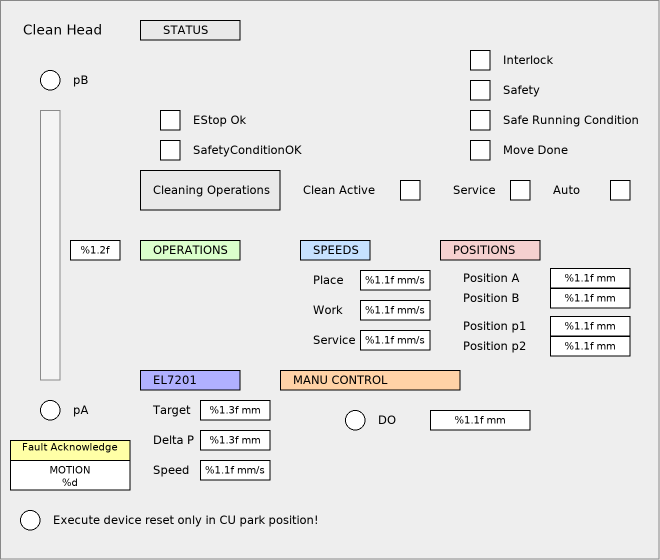
VISUALIZATION _VISU_CLEAN_CH  // 660x560
VAR_IN_OUT
  m_Inst : INT;               (*visu instance*) 
END_VAR
    Rectangle (0,0 660x560)
    Polyline (210,380)
    Polyline (510,250)
    Polyline (300,250)
    Rectangle (280,370 180x20)
    Rectangle (300,240 70x20)
    Rectangle (440,240 100x20)
    Rectangle (140,240 100x20)
    Rectangle (70,400 40x20), "pA"
    Ellipse (40,400 20x20), colour toggle: PRG_MACHINE.fb_CleaningCH[m_Inst].bL_Sensor_pA
    Ellipse (40,70 20x20), colour toggle: PRG_MACHINE.fb_CleaningCH[m_Inst].bI_Sensor_pB
    Rectangle (70,70 50x20), "pB"
    Rectangle (70,240 50x20), "%1.2f", text variable: 1000 * PRG_MACHINE.fb_CleaningCH[m_Inst].fB_Axis.fO_ActualPosition
    Rectangle (375,410 40x20), "DO"
    Rectangle (290,370 170x20), "MANU CONTROL"
    Polyline (450,380)
    Rectangle (310,240 70x20), "SPEEDS"
    Rectangle (360,270 70x20), "%1.1f mm/s", text variable: PRG_MACHINE.fb_CleaningCH[m_Inst].sI_SpeedDef.fP_PlaceSpeed
        OnMouseDown: write the text variable via VisuDialogs.Numpad
    Rectangle (360,300 70x20), "%1.1f mm/s", text variable: PRG_MACHINE.fb_CleaningCH[m_Inst].sI_SpeedDef.fP_WorkSpeed
        OnMouseDown: write the text variable via VisuDialogs.Numpad
    Rectangle (360,330 70x20), "%1.1f mm/s", text variable: PRG_MACHINE.fb_CleaningCH[m_Inst].sI_SpeedDef.fP_ServiceSpeed
        OnMouseDown: write the text variable via VisuDialogs.Numpad
    Rectangle (310,270 60x20), "Place"
    Rectangle (310,300 60x20), "Work"
    Rectangle (310,330 60x20), "Service"
        OnMouseDown: write the text variable via Edit
    Rectangle (550,268 80x20), "%1.1f mm", text variable: PRG_MACHINE.fb_CleaningCH[m_Inst].fI_Position_A
        OnMouseDown: write the text variable via VisuDialogs.Numpad
    Rectangle (460,268 85x20), "Position A"
    Rectangle (460,288 85x20), "Position B"
    Rectangle (550,288 80x20), "%1.1f mm", text variable: PRG_MACHINE.fb_CleaningCH[m_Inst].fI_Position_B
        OnMouseDown: write the text variable via VisuDialogs.Numpad
    Rectangle (450,240 90x20), "POSITIONS"
    Polyline (210,250)
    Rectangle (150,240 90x20), "OPERATIONS"
    Scrollbar (40,110 20x270)
        p3598130195: PRG_MACHINE.sADS_CleanAxis[iCPr_MAP_Cp_ChAxis[m_Inst]].sO_AxisPosition.fC_Min
        p2245068023: PRG_MACHINE.sADS_CleanAxis[iCPr_MAP_Cp_ChAxis[m_Inst]].sO_AxisPosition.fC_Max
        p1057716461: PRG_MACHINE.fb_CleaningCH[m_Inst].fB_Axis.fO_ActualPosition * 1000
    Ellipse (345,410 20x20), colour toggle: PRG_MACHINE.sADS_CleanAxis[iCPr_MAP_Cp_ChAxis[m_Inst]].bI_ManualMove, input disabled if: NOT PRG_MACHINE.sADS_CleanAxis[iCPr_MAP_Cp_ChAxis[m_Inst]].bO_ManualMoveCanEx
        toggle PRG_MACHINE.sADS_CleanAxis[iCPr_MAP_Cp_ChAxis[m_Inst]].bI_ManualMove
    Rectangle (20,20 120x20), "Clean Head"
    Rectangle (140,370 100x20)
    Rectangle (150,460 70x20), "Speed"
    Rectangle (200,460 70x20), "%1.1f mm/s", text variable: 1000 * PRG_MACHINE.fb_CleaningCH[m_Inst].fB_Axis.fI_SpeedLimit
    Rectangle (150,370 90x20), "EL7201"
    Rectangle (10,440 120x50), "Fault Acknowledge", colour toggle: (PRG_MACHINE.fb_CleaningCH[m_Inst].wL_ErrorCode) <> 0
    Polyline (130,450)
    RoundedRectangle (10,460 120x30), "%d", text variable: PRG_MACHINE.fb_CleaningCH[m_Inst].wL_ErrorCode
        tap PRG_MACHINE.sADS_CleanAxis[iCPr_MAP_Cp_ChAxis[m_Inst]].bI_FaultAck
    RoundedRectangle (40,460 60x20), "MOTION"
    Rectangle (140,170 140x40)
    Rectangle (140,20 100x20)
    Polyline (140,30)
    Polyline (240,30)
    Rectangle (160,20 60x20), "STATUS"
    RoundedRectangle (160,110 20x20), colour toggle: PRG_MACHINE.bL_IO_EStopOK
    RoundedRectangle (160,140 20x20), colour toggle: PRG_MACHINE.fB_Machine.bI_SafetyOk
    RoundedRectangle (470,140 20x20), colour toggle: NOT PRG_MACHINE.fb_CleaningCH[m_Inst].bL_Busy
    Rectangle (190,110 120x20), "EStop Ok"
    Rectangle (190,140 120x20), "SafetyConditionOK"
    Rectangle (500,140 90x20), "Move Done"
    RoundedRectangle (470,80 20x20), colour toggle: PRG_MACHINE.fb_CleaningCH[m_Inst].bI_SafeToMove
    Rectangle (500,80 120x20), "Safety"
    RoundedRectangle (470,50 20x20), colour toggle: PRG_MACHINE.fb_CleaningCH[m_Inst].bI_SafeToMove
    Rectangle (500,50 120x20), "Interlock"
    Polyline (650,160)
    Rectangle (150,180 140x20), "Cleaning Operations"
    Polyline (280,200)
    RoundedRectangle (470,110 20x20), colour toggle: PRG_MACHINE.fb_CleaningCH[m_Inst].bL_SafeRunningCondition
    Rectangle (500,110 150x20), "Safe Running Condition"
    RoundedRectangle (610,180 20x20), colour toggle: PRG_MACHINE.fb_CleanProcess[m_Inst].bI_UsrAutoMode
    Rectangle (550,180 60x20), "Auto"
    Polyline (350,80)
    RoundedRectangle (510,180 20x20), colour toggle: PRG_MACHINE.fb_CleanProcess[m_Inst].bI_UsrService
    Rectangle (450,180 60x20), "Service"
    Rectangle (300,180 90x20), "Clean Active"
    RoundedRectangle (400,180 20x20), colour toggle: PRG_MACHINE.fb_CleanProcess[m_Inst].fB_StateCleaning.bL_DevOpActive
    Rectangle (200,400 70x20), "%1.3f mm", text variable: 1000 * PRG_MACHINE.fb_CleaningCH[m_Inst].fB_Axis.fI_TargetPosition
    Rectangle (150,400 70x20), "Target"
    Rectangle (150,430 70x20), "Delta P"
    Rectangle (200,430 70x20), "%1.3f mm", text variable: 1000 * PRG_MACHINE.fb_CleaningCH[m_Inst].fB_Axis.fL_Delta_P
    Rectangle (430,410 100x20), "%1.1f mm", text variable: PRG_MACHINE.sADS_CleanAxis[iCPr_MAP_Cp_ChAxis[m_Inst]].fI_ManualTargetPos
        OnMouseDown: write the text variable via VisuDialogs.Numpad, min PRG_MACHINE.fb_CleaningCH[m_Inst].fI_Position_A, max PRG_MACHINE.fb_CleaningCH[m_Inst].fI_Position_B
    Rectangle (550,316 80x20), "%1.1f mm", text variable: PRG_MACHINE.fb_CleaningCH[m_Inst].fI_Position_p1
        OnMouseDown: write the text variable via VisuDialogs.Numpad
    Rectangle (460,316 85x20), "Position p1"
    Rectangle (460,336 85x20), "Position p2"
    Rectangle (550,336 80x20), "%1.1f mm", text variable: PRG_MACHINE.fb_CleaningCH[m_Inst].fI_Position_p2
        OnMouseDown: write the text variable via VisuDialogs.Numpad
    Ellipse (20,510 20x20), colour toggle: PRG_MACHINE.fb_CleaningCH[m_Inst].bIDp_DeviceReset, input disabled if: NOT PRG_MACHINE.fb_CleaningCU[m_Inst].pInPosCappingClean
        tap PRG_MACHINE.fb_CleaningCH[m_Inst].bIDp_DeviceReset
    Rectangle (50,510 306x20), "Execute device reset only in CU park position!"
END_VISUALIZATION

(* stored: Version 1.1.0.1, ProductVersion 3.1.4024.9
   Visu _VISU_CLEAN_CH: Id {fd35c074-71b6-4678-9fe3-93169c9b195e} *)
